# EPICS substitutions: vacuum/MAIN_TRUNK/vacApp/Db/l210_agilent4uhv.substitutions
# Agilent4UHV substitutions file

file db/agilent4uhv.db
{
     pattern {LOCA,			DEV,			PORT,		ADDR,	TIMEOUT}
     		 {HL2,			VL210_1,		4uhv_1,		0,		0.2}
     		 {HL2,			VL210_2,		4uhv_2,		0,		0.2}
}
file db/agilent4uhv_alias.db
{
     pattern {LOCA,			DEV,		SUB1,					SUB2,					SUB3,						SUB4,				PORT,       ADDR,   TIMEOUT}
     		 {HL2,			VL210_1,	IP01:L210_Acc601,		IP02:L210_Acc602,		IP03:L210_Acc603,			IP04:L210_Acc604,	4uhv_1,     0,      0.2}
     		 {HL2,			VL210_2,	IP05:L210_Acc605,		IP06:L210_Wave601,		IP07:L210_Kly601,			IP08:NOTUSED,		4uhv_1,     0,      0.2}
}
